(* IEC 61131-3 sources: tfc-hmi/packages/tfc_mcp_server/test/compiler/fixtures/schneider, 2 files *)

(* ---- direct_addressing.st ---- *)
PROGRAM SchneiderIO
VAR
  motorStart AT %I0.3.5 : BOOL;
  motorRun AT %Q0.4.0 : BOOL;
  speedCmd AT %MW100 : INT;
  tempSensor AT %IW0.2.0 : INT;
  internalBit AT %M200 : BOOL;
  internalWord AT %MW500 : INT;
END_VAR
  IF motorStart THEN
    motorRun := TRUE;
    speedCmd := 1500;
  ELSE
    motorRun := FALSE;
    speedCmd := 0;
  END_IF;

  // Direct address in expression
  %MW101 := %MW100 + 1;
  IF %I0.3.6 THEN
    %Q0.4.1 := TRUE;
  END_IF;
END_PROGRAM

(* ---- ebool_types.st ---- *)
PROGRAM SchneiderTypes
VAR
  startButton : EBOOL;
  stopButton : EBOOL;
  motorStatus : EBOOL;
  alarmWord : WORD;
  speedRef : REAL;
  myString : STRING[32] := 'Hello World';
END_VAR
  IF startButton AND NOT stopButton THEN
    motorStatus := TRUE;
    speedRef := 50.0;
  ELSE
    motorStatus := FALSE;
    speedRef := 0.0;
  END_IF;
END_PROGRAM
